{attribute 'linkalways'}
{attribute 'no_explicit_call' := 'do not call this POU directly'}
{attribute 'enable_dynamic_creation'}
FUNCTION_BLOCK ABSTRACT JsonPathElement EXTENDS Disposable IMPLEMENTS I_JsonPathElement
VAR
	_previousElement, _nextElement : I_JsonPathElement;
END_VAR

METHOD AddReference
VAR_INPUT
END_VAR
IF NextElement <> 0 THEN
	NextElement.AddReference();
END_IF

SUPER^.AddReference();
END_METHOD

METHOD FB_init : BOOL
VAR_INPUT
	bInitRetains : BOOL; // if TRUE, the retain variables are initialized (warm start / cold start)
	bInCopyCode : BOOL;  // if TRUE, the instance afterwards gets moved into the copy code (online change)
	PreviousElement : I_JsonPathElement;
	NextElement : I_JsonPathElement; 
END_VAR
THIS^._previousElement := PreviousElement;
THIS^._nextElement := NextElement;
END_METHOD

PROPERTY PUBLIC NextElement : I_JsonPathElement
GET
NextElement := _nextElement;
END_GET
SET
VAR
	self : I_JsonPathElement;
END_VAR
_nextElement := NextElement;

IF NextElement = 0 THEN
	RETURN;
END_IF

self := THIS^;

IF NextElement.PreviousElement <> self THEN
	NextElement.PreviousElement := self;
END_IF;
END_SET
END_PROPERTY

PROPERTY PUBLIC PreviousElement : I_JsonPathElement
GET
PreviousElement := _previousElement;
END_GET
SET
VAR
	self : I_JsonPathElement;
END_VAR
_previousElement := PreviousElement;

IF PreviousElement = 0 THEN
	RETURN;
END_IF

self := THIS^;

IF PreviousElement.NextElement <> self THEN
	PreviousElement.NextElement := self;
END_IF;
END_SET
END_PROPERTY

PROPERTY PUBLIC ABSTRACT PropertyName : T_MAXSTRING
GET
END_GET
END_PROPERTY

METHOD Release
VAR_INPUT
END_VAR
IF PreviousElement <> 0 THEN
	PreviousElement.NextElement := 0;
	PreviousElement.Release();
END_IF

IF NextElement <> 0 THEN
	NextElement.PreviousElement := 0;
	NextElement.Release();
END_IF

SUPER^.Release();
END_METHOD

METHOD PUBLIC ABSTRACT ResolveToSJsonValue : SJsonValue
VAR_INPUT
	jsonParser : REFERENCE TO FB_JsonDomParser;
	jsonDocument : SJsonValue;
END_VAR
END_METHOD

END_FUNCTION_BLOCK

(* stored: Version 1.1.0.1, ProductVersion 3.1.4024.12
   POU JsonPathElement: Id {8edb91a2-c526-4ba3-97c5-b8729709b0f1}, SpecialFunc None
   Folder Constructor: Id {7c5d3272-7068-4e31-9308-ece34c233939}
   Method AddReference: Id {dad9e4ce-73ab-4ec4-8485-a9fd7782fc44}
   Method FB_init: Id {a183be44-c225-4cef-8331-2a267a1d3ac0}
   Property NextElement: Id {d7414643-0085-464a-8aaa-7fc8dec9e8c5}
   Get Get: Id {11ed51b8-db1a-4170-9d56-5108ce43f29a}
   Set Set: Id {6b6a0943-9463-4deb-bc4c-a6e9919b5673}
   Property PreviousElement: Id {fa8e8155-b073-46f1-ba1a-e678f9f8631c}
   Get Get: Id {b7d7ff7a-d413-44c3-a2f1-abc277418553}
   Set Set: Id {1fc9578e-d39c-4296-8b48-feab273cc71a}
   Property PropertyName: Id {b1e9ed71-ff90-45f5-aa72-97ff47e73a18}
   Get Get: Id {6e35132e-2626-4816-bfa4-085702aa1d28}
   Method Release: Id {b4a96398-d179-487d-a66a-484379c24608}
   Method ResolveToSJsonValue: Id {f0bbbf78-1f59-4094-be0e-9504726a2ca5} *)
